Staubli VAL3: CopyStrArray.pgx

public program CopyStrArray(string& x_sStrIn[], string& x_sStrOut[])
  local num i
begin
  //复制字符串数组
  while size(x_sStrOut)>1
    delete(x_sStrOut[0])
  endWhile
  x_sStrOut[0]=""
  while x_sStrIn[i]!=""
    x_sStrOut[i]=x_sStrIn[i]
  endWhile
end
